Staubli VAL3: repeat.pgx

public program repeat(num& x_nInput[], num x_nTimes, num& x_nResult[])
  local num l_nElement
  local num l_nTimes
  local num l_nCounter
  local num l_nAppend
begin

  //rep(c(1,2,3),4) -> 1,2,3,1,2,3,1,2,3,1, 2, 3
  //                   0,1,2,3,4,5,6,7,8,9,10,11

  resize(x_nResult,1,size(x_nInput)*x_nTimes)

  for l_nElement = 1 to x_nTimes
    for l_nAppend = 0 to size(x_nInput)-1
      x_nResult[l_nCounter+l_nAppend] = x_nInput[l_nAppend]
    endFor
    l_nCounter = l_nCounter+size(x_nInput)
  endFor


end
